(* CODESYS project contadores111.project
   CustomField01_name: CustomField01
   CustomField08_name: CustomField08
   CustomField06_name: CustomField06
   Title: ATV_IMC_Template
   CustomField09_name: CustomField09
   CustomField07_name: CustomField07
   CustomField05_name: CustomField05
   CustomField02_name: CustomField02
   Description: This template can be used for a correct interface with the local drive. the MANDATORY_AT_EACH_CYCLE program must be called like it is done in this application.
   CustomField04_name: CustomField04
   CustomField10_name: CustomField10
   Version: 0.0.0.0
   Company: Schneider Electric
   CustomField03_name: CustomField03

Project tree, tasks and I/O mapping:
  MyController : TM241CE24R, Schneider Electric, order no. TM241CE24R, version 4.0.2.9
    application Application
      task MAST (cyclic, interval 20 ms, priority 15, watchdog 100 ms x 1) calls temporizadores
      function HiddenPOU [ST]
      global variables GVL
      program temporizadores [LD]
    DI : Digital Inputs, Schneider Electric, version 4.0.2.9
        input  iwDI_IW0 : WORD  // IW0
        input  ibDI_IB1 : BYTE  // IB1
    DQ : Digital Outputs, Schneider Electric, version 4.0.2.9
        output qwDQ_QW0 : WORD  // QW0
        output qbDQ_QB1 : BYTE  // QB1
    Counters : Counters, Schneider Electric, version 4.0.2.9
    Pulse_Generators : Pulse Generators, Schneider Electric, version 4.0.2.9
    Cartridge_1 : Cartridge, Schneider Electric, version 4.0.2.9
    IO_Bus : IO bus - TM3, Schneider Electric, version 4.0.2.9
    COM_Bus : COM bus, Schneider Electric, version 4.0.2.9
    Ethernet_1 : Ethernet Network, Schneider Electric, version 4.0.2.9
    Serial_Line_1 : Serial line, Schneider Electric, version 4.0.2.9
      SoMachine_Network_Manager : SoMachine-Network Manager, Schneider Electric, version 4.0.0.2
    Serial_Line_2 : Serial line, Schneider Electric, version 4.0.2.9
      Modbus_Manager : Modbus Manager, Schneider Electric, version 4.0.0.2
  text list GlobalTextList
  GlobalImagePool
*)

// MyController/Application/GVL
VAR_GLOBAL
	// este es el pulsador de marcha
	marcha: BOOL;
END_VAR

// MyController/Application/temporizadores
PROGRAM temporizadores
VAR
	m1: BOOL;
	CTUD_0: CTUD;
	sensalida: BOOL;
	reset: BOOL;
	load: BOOL;
	contacoche: CTUD;
	sensentrada: BOOL;
	lverde: BOOL;
	lambar: BOOL;
	limiteuser: INT;
	lroja: BOOL;
END_VAR

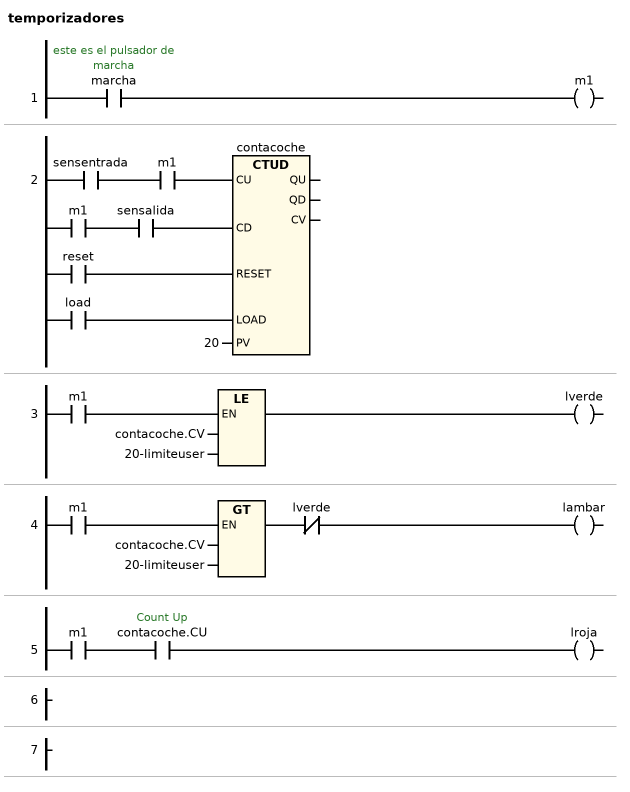
// NETWORK 1
//   marcha: este es el pulsador de marcha
m1 := marcha;

// NETWORK 2
contacoche(CU := sensentrada AND m1, CD := m1 AND sensalida, RESET := reset, LOAD := load, PV := 20); // CTUD

// NETWORK 3
//   contacoche.CV: Current Counter Value
lverde := m1 AND contacoche.CV <= (20-limiteuser);

// NETWORK 4
//   contacoche.CV: Current Counter Value
lambar := (m1 AND contacoche.CV > (20-limiteuser)) AND NOT lverde;

// NETWORK 5
//   contacoche.CU: Count Up
lroja := m1 AND contacoche.CU;

// NETWORK 6

// NETWORK 7

END_PROGRAM

// MyController/Application/HiddenPOU
FUNCTION HiddenPOU : BOOL

VAR_INPUT
	pHiddenFunc: POINTER TO WORD;
END_VAR
VAR
	pRead: POINTER TO BYTE;
	pWrite: POINTER TO BYTE;
END_VAR

pRead := pHiddenFunc + 400;
pWrite := pHiddenFunc + 4400;
HiddenPOU := TRUE;

END_FUNCTION
